{attribute 'qualified_only'}
{attribute 'analysis' := '-33'}
VAR_GLOBAL
	MonitorTestData		: MonitorTest;
	ReadTestData		: ReadTest;
	SymbolTestData		: SymbolTest;
	WriteTestData		: WriteTest;
END_VAR

(* stored: Version 1.1.0.1, ProductVersion 3.1.4024.12
   GVL Ads: Id {40635e17-4a82-430d-a3a9-4285c5608b90} *)
